SYSTEM simpleAlphabot
  (* Version 1.0, 2023-01-19, test *)
  APPLICATION simpleAlphabotApp
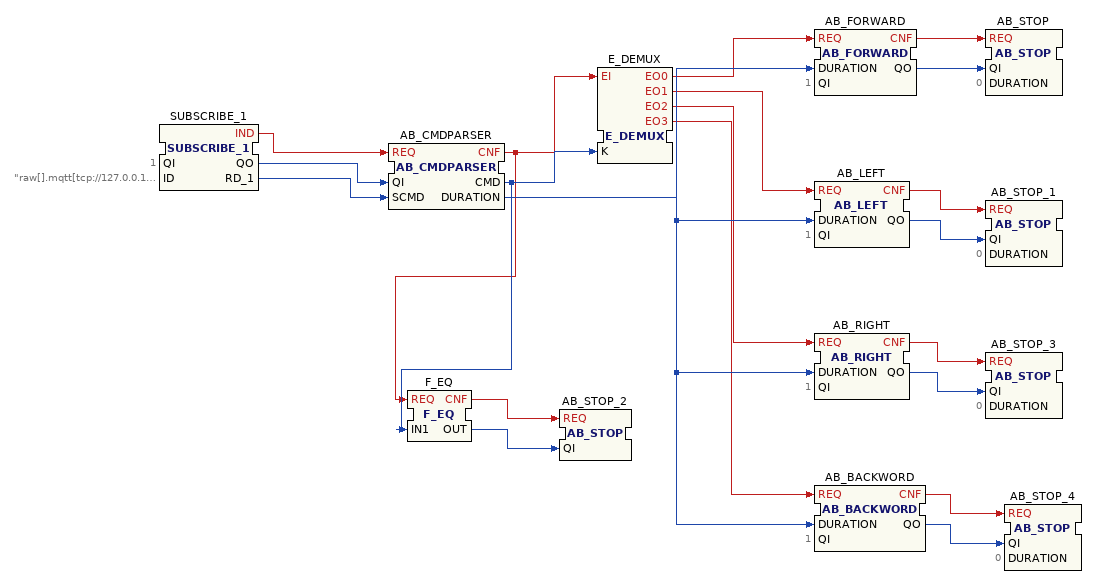
    FBS
      SUBSCRIBE_1 : SUBSCRIBE_1(QI := 1, ID := "raw[].mqtt[tcp://127.0.0.1:1883, abot, abto_cmd]");
      AB_CMDPARSER : AB_CMDPARSER;
      AB_BACKWORD : AB_BACKWORD(QI := 1);
      AB_FORWARD : AB_FORWARD(QI := 1);
      AB_STOP : AB_STOP(DURATION := 0);
      E_DEMUX : E_DEMUX;
      AB_LEFT : AB_LEFT(QI := 1);
      AB_RIGHT : AB_RIGHT(QI := 1);
      AB_STOP_1 : AB_STOP(DURATION := 0);
      AB_STOP_2 : AB_STOP;
      F_EQ : F_EQ;
      AB_STOP_3 : AB_STOP(DURATION := 0);
      AB_STOP_4 : AB_STOP(DURATION := 0);
    END_FBS
    EVENT_CONNECTIONS
      SUBSCRIBE_1.IND TO AB_CMDPARSER.REQ;
      AB_FORWARD.CNF TO AB_STOP.REQ;
      AB_CMDPARSER.CNF TO F_EQ.REQ;
      F_EQ.CNF TO AB_STOP_2.REQ;
      AB_CMDPARSER.CNF TO E_DEMUX.EI;
      E_DEMUX.EO0 TO AB_FORWARD.REQ;
      E_DEMUX.EO1 TO AB_LEFT.REQ;
      E_DEMUX.EO2 TO AB_RIGHT.REQ;
      AB_BACKWORD.CNF TO AB_STOP_4.REQ;
      AB_RIGHT.CNF TO AB_STOP_3.REQ;
      AB_LEFT.CNF TO AB_STOP_1.REQ;
      E_DEMUX.EO3 TO AB_BACKWORD.REQ;
    END_CONNECTIONS
    DATA_CONNECTIONS
      SUBSCRIBE_1.QO TO AB_CMDPARSER.QI;
      SUBSCRIBE_1.RD_1 TO AB_CMDPARSER.SCMD;
      AB_FORWARD.QO TO AB_STOP.QI;
      AB_CMDPARSER.CMD TO F_EQ.IN1;
      F_EQ.OUT TO AB_STOP_2.QI;
      AB_CMDPARSER.CMD TO E_DEMUX.K;
      AB_CMDPARSER.DURATION TO AB_FORWARD.DURATION;
      AB_CMDPARSER.DURATION TO AB_LEFT.DURATION;
      AB_CMDPARSER.DURATION TO AB_RIGHT.DURATION;
      AB_CMDPARSER.DURATION TO AB_BACKWORD.DURATION;
      AB_BACKWORD.QO TO AB_STOP_4.QI;
      AB_RIGHT.QO TO AB_STOP_3.QI;
      AB_LEFT.QO TO AB_STOP_1.QI;
    END_CONNECTIONS
  END_APPLICATION
END_SYSTEM
